{attribute 'qualified_only'}
VAR_GLOBAL
	bAuto		: BOOL;
	bRunning	: BOOL;
END_VAR

(* stored: Version 1.1.0.1
   GVL GVL: Id {d563e694-ff00-46c8-af8a-4927b3fd6f89} *)
